VISUALIZATION HMI  // 2x2
END_VISUALIZATION

(* stored: Version 1.1.0.1, ProductVersion 3.1.4024.12
   Visu HMI: Id {194792d2-46fe-405f-bf6e-7c6c6a84345e} *)
